// Mitsubishi GX Works2 project: ACMotor   PLC: Q03UD

PROGRAM MAIN
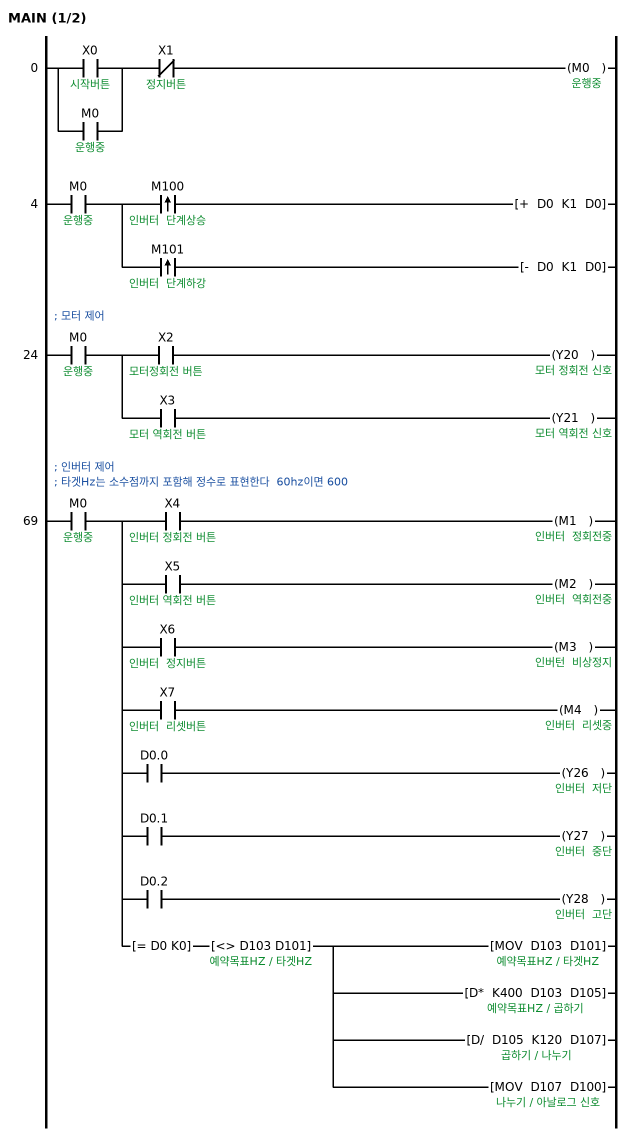
0     LD      X0  ; 시작버튼
      OR      M0  ; 운행중
      ANI     X1  ; 정지버튼
      OUT     M0  ; 운행중
4     LD      M0  ; 운행중
      MPS
      ANDP    M100  ; 인버터  단계상승
      +       D0 K1 D0
      MPP
      ANDP    M101  ; 인버터  단계하강
      -       D0 K1 D0
; 모터 제어
24    LD      M0  ; 운행중
      MPS
      AND     X2  ; 모터정회전 버튼
      OUT     Y20  ; 모터 정회전 신호
      MPP
      AND     X3  ; 모터 역회전 버튼
      OUT     Y21  ; 모터 역회전 신호
; 인버터 제어
; 타겟Hz는 소수점까지 포함해 정수로 표현한다  60hz이면 600
69    LD      M0  ; 운행중
      MPS
      AND     X4  ; 인버터 정회전 버튼
      OUT     M1  ; 인버터  정회전중
      MRD
      AND     X5  ; 인버터 역회전 버튼
      OUT     M2  ; 인버터  역회전중
      MRD
      AND     X6  ; 인버터  정지버튼
      OUT     M3  ; 인버턴  비상정지
      MRD
      AND     X7  ; 인버터  리셋버튼
      OUT     M4  ; 인버터  리셋중
      MRD
      AND     D0.0
      OUT     Y26  ; 인버터  저단
      MRD
      AND     D0.1
      OUT     Y27  ; 인버터  중단
      MRD
      AND     D0.2
      OUT     Y28  ; 인버터  고단
      MPP
      AND=    D0 K0
      AND<>   D103 D101  ; 예약목표HZ / 타겟HZ
      MOV     D103 D101
      D*      K400 D103 D105  ; 곱하기
      D/      D105 K120 D107  ; 나누기
      MOV     D107 D100  ; 아날로그 신호
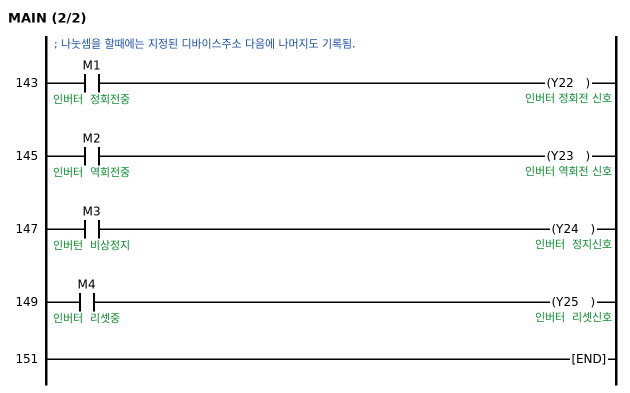
; 나눗셈을 할때에는 지정된 디바이스주소 다음에 나머지도 기록됨.
143   LD      M1  ; 인버터  정회전중
      OUT     Y22  ; 인버터 정회전 신호
145   LD      M2  ; 인버터  역회전중
      OUT     Y23  ; 인버터 역회전 신호
147   LD      M3  ; 인버턴  비상정지
      OUT     Y24  ; 인버터  정지신호
149   LD      M4  ; 인버터  리셋중
      OUT     Y25  ; 인버터  리셋신호
151   END
END_PROGRAM

// device comments not shown above
D1  ; 인버터  타겟Hz
D2  ; 인버터  예약Hz
D3  ; 곱하기 저장
D4  ; 곱하기 저장
D5  ; 나눗셈 저장
D6  ; 나누기 저장
